/// This enumeration contains all steps that are used by the various sequences of a unit.
/// Sequences use a subrange (***Begin to ***End) of this enumeration.
{attribute 'qualified_only'}
{attribute 'to_string'}
TYPE TransportStep :
(
  Undefined := 0
  
  ,BootBegin
  ,BootEnd 

  ,StopBegin
  ,StopEnd

  ,AutomaticBegin
  ,AutomaticInitializeMovements  
  ,AutomaticMoveToLeftPos
  ,AutomaticWaitSomeTime
  ,AutomaticMoveVerticalDown
  ,AutomaticCloseGripper
  ,AutomaticMoveVerticalToTopPos  
  ,AutomaticWaitSomeMoreTime
  ,AutomaticMoveToRightPos
  ,AutomaticCleanUp
  ,AutomaticOpenGripper
  ,AutomaticMoveToCamPos
  ,AutomaticStartQualityInspection
  ,AutomaticEnd
  
  ,GoHomeBegin
  ,GoHomeStartHomingOfChilds
  ,GoHomeVerticalUp
  ,GoHomeHorizontalToRightPos
  ,GoHomeUnlockQualityInspection
  ,GoHomeEnd 
  
  ,FaultReactionBegin
  ,FaultReactionVerticalUp
  ,FaultReactionEnd
);
END_TYPE

(* stored: Version 1.1.0.1
   DUT TransportStep: Id {0156a6d2-d3bb-4b09-8f1f-ec928c6b4e4b} *)
